// TIA Portal project "2020-10-23_StartStopMotore" (V16)

(* hardware
DEVICE "S7-1200 station_1"  S7-1200 Station
   slot 0: "Telaio di montaggio_0"  Rack  V1.0
   slot 1: "PLC_1"  CPU 1215C DC/DC/DC  6ES7 215-1AG40-0XB0  V4.2
*)

// ===== PLC "PLC_1"  CPU 1215C DC/DC/DC =====

VAR_GLOBAL   // PLC tag table "Tabella delle variabili standard"
   "Vent_A_NA" AT %I0.0 : Bool;
   "Vent_B_NA" AT %I0.1 : Bool;
   "Vent_C_NA" AT %I0.2 : Bool;
   "Start_NA" AT %I0.3 : Bool;
   "Stop_NA" AT %I0.4 : Bool;
   "Allarme_NA" AT %I0.5 : Bool;
   "Ripristino_NA" AT %I0.6 : Bool;
   "In7" AT %I0.7 : Bool;
   "Motore" AT %Q0.0 : Bool;
   "Vent_2su3_OK" AT %Q0.1 : Bool;
   "Allarme_mem" AT %M0.0 : Bool;
END_VAR

ORGANIZATION_BLOCK "Main"   // OB1, LAD, ProgramCycle
TITLE = "Main Program Sweep (Cycle)"
{ S7_Optimized_Access := 'TRUE' }
VERSION : 0.1
// Gestione di un motore, con almeno 2 ventilatori su 3 che funzionano e un allarme con memorizzazione ripristino e rientro
// I0.0, Vent_A, NA
// I0.1, Vent_B, NA
// I0.2, Vent_C, NA
// I0.3, Start, NA
// I0.4, Stop, NA
// I0.5 Allarme, NA
// I0.6 Ripristino, NA
// 
// Q0.0 Motore
// Q0.1 Ventilazione OK (almeno 2 ventilatori su 3 sono in funzione)
// 
// M0.0 Allarme memorizzato (Lampada di allarme)
BEGIN

REGION Network 1: Gestione Vent_OK
   // Uso la bobina perchè gestisco questa uscita solo in questo segmento
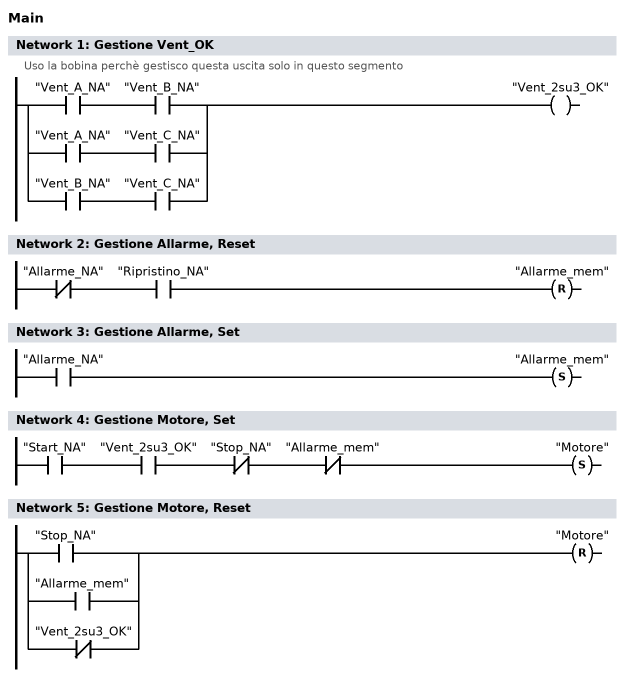
   RUNG wire#powerrail
      Contact( "Vent_A_NA" )
      Contact( "Vent_B_NA" )
      wire#w1
      Coil( "Vent_2su3_OK" )
   END_RUNG
   RUNG wire#powerrail
      Contact( "Vent_A_NA" )
      Contact( "Vent_C_NA" )
   END_RUNG wire#w1
   RUNG wire#powerrail
      Contact( "Vent_B_NA" )
      Contact( "Vent_C_NA" )
   END_RUNG wire#w1
   // the same network as SCL:
   "Vent_2su3_OK" := ("Vent_A_NA" AND "Vent_B_NA") OR ("Vent_A_NA" AND "Vent_C_NA") OR ("Vent_B_NA" AND "Vent_C_NA");
END_REGION

REGION Network 2: Gestione Allarme, Reset
   RUNG wire#powerrail
      I_Contact( "Allarme_NA" )
      Contact( "Ripristino_NA" )
      R_Coil( "Allarme_mem" )
   END_RUNG
   // the same network as SCL:
   IF NOT "Allarme_NA" AND "Ripristino_NA" THEN "Allarme_mem" := FALSE; END_IF;
END_REGION

REGION Network 3: Gestione Allarme, Set
   RUNG wire#powerrail
      Contact( "Allarme_NA" )
      S_Coil( "Allarme_mem" )
   END_RUNG
   // the same network as SCL:
   IF "Allarme_NA" THEN "Allarme_mem" := TRUE; END_IF;
END_REGION

REGION Network 4: Gestione Motore, Set
   RUNG wire#powerrail
      Contact( "Start_NA" )
      Contact( "Vent_2su3_OK" )
      I_Contact( "Stop_NA" )
      I_Contact( "Allarme_mem" )
      S_Coil( "Motore" )
   END_RUNG
   // the same network as SCL:
   IF "Start_NA" AND "Vent_2su3_OK" AND NOT "Stop_NA" AND NOT "Allarme_mem" THEN "Motore" := TRUE; END_IF;
END_REGION

REGION Network 5: Gestione Motore, Reset
   RUNG wire#powerrail
      Contact( "Stop_NA" )
      wire#w1
      R_Coil( "Motore" )
   END_RUNG
   RUNG wire#powerrail
      Contact( "Allarme_mem" )
   END_RUNG wire#w1
   RUNG wire#powerrail
      I_Contact( "Vent_2su3_OK" )
   END_RUNG wire#w1
   // the same network as SCL:
   IF "Stop_NA" OR "Allarme_mem" OR NOT "Vent_2su3_OK" THEN "Motore" := FALSE; END_IF;
END_REGION
END_ORGANIZATION_BLOCK